// Code généré automatiquement : NE PAS MODIFIER
FUNCTION CheckBounds : DINT
VAR_INPUT
	index, lower, upper: DINT;
END_VAR

// Code généré automatiquement : Il s’agit d’une proposition d’implémentation.
{noflow}
Fault_Count_G(CU:=FALSE) ; 
IF  index < lower THEN
	CheckBounds := lower;
	Fault_Count_G(CU:=TRUE) ; 
ELSIF  index > upper THEN
	CheckBounds := upper;
	Fault_Count_G(CU:=TRUE) ; 
ELSE  
	CheckBounds := index;
END_IF
{flow}

END_FUNCTION

(* stored: Version 1.1.0.1, ProductVersion 3.1.4024.6
   POU CheckBounds: Id {a0070896-dbd0-4dbe-a242-7361e1e52187}, SpecialFunc CheckBounds *)
